{attribute 'GeneratedUsingTerminal: EP6001-0002-0020'}
{attribute addProperty BoxType "EP6001-0002-0020"}
{attribute addProperty Id "StatusAT %I*UINT2Data_InAT %I*ARRAY[0..21] OF USINT22"}
{attribute addProperty CRC "1367962124"}
{attribute addProperty Size "24"}
TYPE COM_Inputs_6C2FC202 :
STRUCT
	{attribute addProperty Name "Status"}
	Status AT %I* : UINT;
	{attribute addProperty Name "Data_In"}
	Data_In AT %I* : ARRAY[0..21] OF USINT;
END_STRUCT
END_TYPE

(* stored: Version 1.2.0.0, ProductVersion 3.1.4024.9
   DUT COM_Inputs_6C2FC202: Id {470a17f4-ad6d-4ce0-a14e-d6a146a88438} *)
